(* IEC 61131-3 sources: repolevel_ST_code_completion/output/0122完整版本_无planner目前sota/repoeval_measurement_control/readful_result_no_provide, 1 file *)

(* ---- Tank.st ---- *)
VAR
	name								:STRING;
	bLevel								:BOOL;
	bTemp								:BOOL;
END_VAR

name := stName;

IF(nUnitLevel > nMaxLevel) THEN
	bLevel := FALSE;
END_IF
IF(nUnitLevel < nMinLevel) THEN
	bLevel := TRUE;
END_IF

IF(bLevel) THEN
	nUnitLevel := nUnitLevel + 1;
ELSE
	nUnitLevel := nUnitLevel - 1;
END_IF

IF(nUnitTemp > nMaxTemp) THEN
	bTemp := FALSE;
END_IF
IF(nUnitTemp < nMinTemp) THEN
	bTemp := TRUE;
END_IF

IF(bTemp) THEN
	nUnitTemp := nUnitTemp + 1;
ELSE
	nUnitTemp := nUnitTemp - 1;
END_IF
END_FUNCTION_BLOCK
